PROGRAM prgHouse_H1
VAR
	fbHouse				: FB_HouseC_Power_Virtual;
	bHouseEnabled		: BOOL;						//{#lynus.ag#()}
	lrPowerHouse		: LREAL;					//{#lynus.ag#()}
	lrPowerHouse_Manual	: LREAL;					//{#lynus.ag#()}
END_VAR
VAR PERSISTENT
	bEnableHouse		: BOOL;						//{#lynus.ag#()}
END_VAR

fbHouse(
	bEnable:= bEnableHouse, 
	diNrOfEMS_IN:= prgEMS_H1.fbEMS.diNrOfEMS_OUT, 
	bSetDefault:= , 
	lrCounterConsumptionSetDefault:= , 
	lrCounterProductionSetDefault:= , 
	stDataHouseC=> , 
	diNrOfHouseC_OUT=> );
	
bHouseEnabled := fbHouse.stDataHouseC.bEnabled;
lrPowerHouse := fbHouse.stDataHouseC.lrPower;	
lrPowerHouse_Manual := prgPV_H1.lrPowerPV + prgGrid_H1.fbEM1.stDataEMPowerRealTime.lrPowerTotal + prgBattery_H1.lrPowerBattery;

END_PROGRAM

(* stored: Version 1.1.0.1, ProductVersion 3.1.4024.11
   POU prgHouse_H1: Id {1004e12f-88fd-4838-a3c1-f7a079c901cf}, SpecialFunc None *)
